PROGRAM Watering
VAR
	
	trigger:F_TRIG;
	waterTimer:TON;
	waterOn:BOOL;
	dtTime:DT;
	todTime:TOD;

END_VAR


GVL.watertingTime:=DWORD_TO_TIME(GVL.HMIWateringTimeSeconds*1000);//in ms
GVL.watertingStart:=DWORD_TO_TOD((GVL.HMIWateringStartHour*60 + GVL.HMIWateringStartMinute)*60*1000);//also in ms



dtTime:=SYSTEMTIME_TO_DT(GVL.fbLocalSystemTime.systemTime);
todTime:=DT_TO_TOD(dtTime);
waterTimer(PT:=GVL.watertingTime);

IF GVL.wateringDays[GVL.fbLocalSystemTime.systemTime.wDayOfWeek]=TRUE THEN
	IF todTime>=GVL.watertingStart AND todTime<=(GVL.watertingStart+GVL.watertingTime) THEN
		waterOn:=TRUE;
	ELSE
		waterOn:=FALSE;
	END_IF
END_IF

END_PROGRAM

(* stored: Version 1.1.0.1, ProductVersion 3.1.4022.18
   POU Watering: Id {19a66220-0e9e-4f45-bda0-7029e04300f6}, SpecialFunc None *)
